Omron CX-Programmer project 新工程 (CX-Programmer 9.73)

# PLC 新PLC1: CPM2* 

## Global symbols (name address type ; comment)
0.11 BOOL  ; �0网�╈�?w�!
10.02 BOOL  ; �6�镧诜z鼯�u靑
11.01 BOOL  ; $?St$Bk?_#[2] / 粋龠诛�� / 顯�(鰟$?St$Bk?_#[2]
11.13 BOOL  ; �*�{得�逌A� �69
13.04 BOOL  ; 制动
13.05 BOOL  ; �东嚼浯�
13.13 BOOL  ; /站齴遅喵顎^
13.14 BOOL  ; '@� nK瞈�饾y�4
15.07 BOOL  ; 獱^践蒘��揧PB�
1.11 BOOL  ; �膈g�e稞��濨5
25.13 BOOL  ; 
2.07 BOOL  ; 4╖�铴�煙呀腩
31.11 BOOL  ; �愴�搡k賴�$欈]
43.02 BOOL  ; 抆葵`|%���A
4.02 BOOL  ; 啐-�旜��FA
6.01 BOOL  ; 卟_�垤��巻(埨O
6.09 BOOL  ; 蓮7挑��┹茒Q
6.13 BOOL  ; 珴;埗�符�禞�b
AR4.01 BOOL  ; _�/頡骫鹐y�a
LR12.14 BOOL  ; �$_Y般鬻锟絸�>
LR13.11 BOOL  ; 慊纂��}煂l 棝v
LR9.05 BOOL  ; J荦�~Mw�	k

## Program 新程序1 (no task)
; 这个PLC程序实现了一个锰钢生产线的控制系统，应用于钢铁厂的锰钢生产工艺。 / 系统包含启动按钮、停止按钮、手动/自动开关、加热炉温度传感器、轧机压力传感器、冷却水流量传感器。 / 外部执行设备包括加热炉控制、轧机控制、冷却水泵控制、报警灯。 / 系统通过启动按钮触发整个流程，随后激活加热炉控制对锰钢原料进行加热。在加热完成后，系统启动轧机控制对原料进行轧制成型。特别地，加热炉控制和轧机控制不可同时启动，以避免设备间的冲突，确保生产过程平稳进行。按下加热按钮时，激活加热炉控制进行加热。按下轧制按钮时，激活轧机控制进行轧制。轧制完成后，启动冷却水泵控制对钢材进行冷却，并确保相关状态正常。启动按钮按下时，激活冷却水泵控制进行冷却。冷却水流量传感器正常时，维持冷却水泵控制的运行。 / 操作员可以通过手动/自动切换开关选择运行模式。在手动模式下，按下手动模式按钮置位手动模式标志，随后通过按钮控制加热炉控制、轧机控制和冷却水泵控制。在自动模式下，按下自动模式按钮置位自动模式标志，随后通过按钮触发流程。手动模式标志和自动模式标志不可同时置位，以保证模式切换的清晰性和安全性。 / 此外，如果加热炉温度传感器检测到温度超限，报警灯会立即点亮，提示操作员采取措施。加热炉温度传感器检测加热状态时，系统进入准备阶段。异常发生时，报警灯点亮提示操作员。同理，当轧机压力传感器检测到压力超出安全范围时，报警灯也会亮起，确保设备不受损。轧机压力传感器检测轧制状态时，系统继续运行。异常发生时，报警灯点亮提示操作员。系统中使用加热炉启动延时定时器 (TIM001)、轧机启动延时定时器 (TIM002) 和冷却水泵启动延时定时器 (TIM003) 控制流程的时间间隔，避免操作过快导致的故障。任何时候按下停止按钮，系统会停止部分输出，确保紧急情况下的安全。

### Section 段1

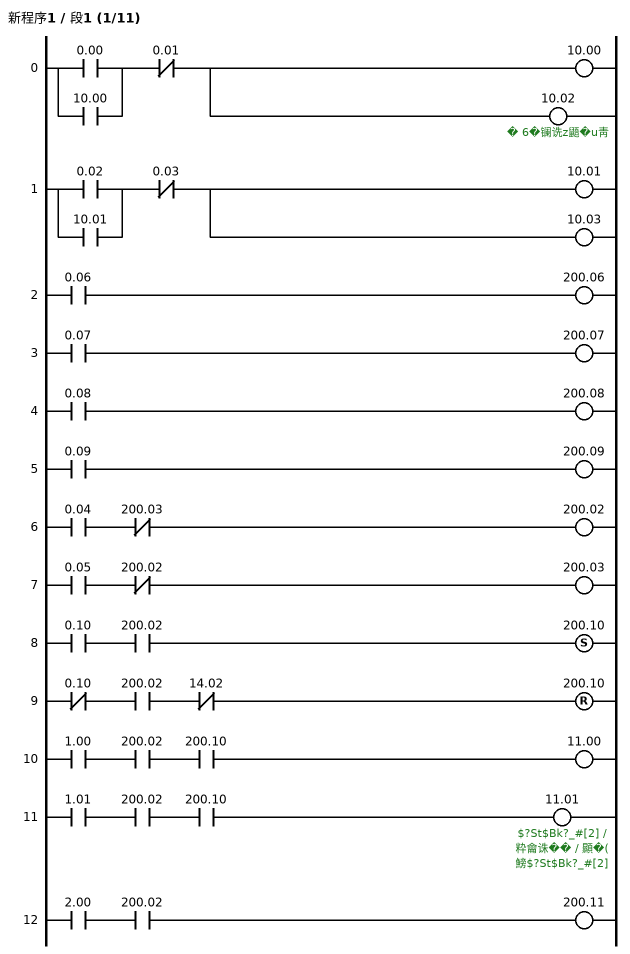
; rung 0
LD 0.00
OR 10.00
ANDNOT 0.01
OUT 10.00
OUT 10.02  ; �6�镧诜z鼯�u靑
; rung 1
LD 0.02
OR 10.01
ANDNOT 0.03
OUT 10.01
OUT 10.03
; rung 2
LD 0.06
OUT 200.06
; rung 3
LD 0.07
OUT 200.07
; rung 4
LD 0.08
OUT 200.08
; rung 5
LD 0.09
OUT 200.09
; rung 6
LD 0.04
ANDNOT 200.03
OUT 200.02
; rung 7
LD 0.05
ANDNOT 200.02
OUT 200.03
; rung 8
LD 0.10
AND 200.02
SET 200.10
; rung 9
LDNOT 0.10
AND 200.02
ANDNOT 14.02
RSET 200.10
; rung 10
LD 1.00
AND 200.02
AND 200.10
OUT 11.00
; rung 11
LD 1.01
AND 200.02
AND 200.10
OUT 11.01  ; $?St$Bk?_#[2] / 粋龠诛�� / 顯�(鰟$?St$Bk?_#[2]
; rung 12
LD 2.00
AND 200.02
OUT 200.11

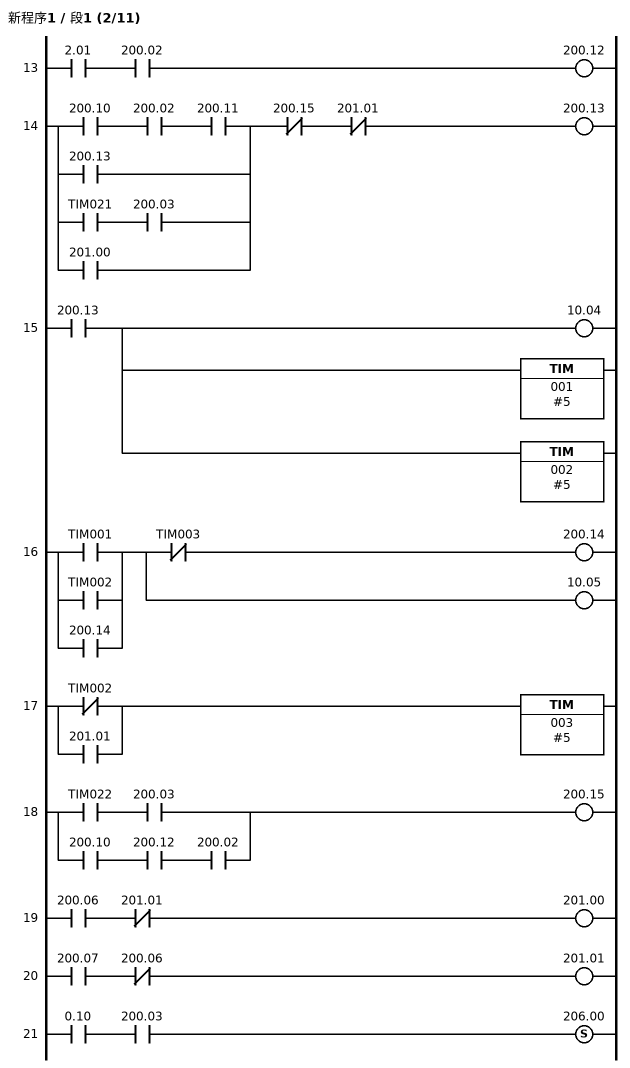
; rung 13
LD 2.01
AND 200.02
OUT 200.12
; rung 14
LD 200.10
AND 200.02
AND 200.11
OR 200.13
LD TIM021
AND 200.03
ORLD
OR 201.00
ANDNOT 200.15
ANDNOT 201.01
OUT 200.13
; rung 15
LD 200.13
OUT 10.04
TIM 001 #5
TIM 002 #5
; rung 16
LD TIM001
OR TIM002
OR 200.14
OUT TR0
ANDNOT TIM003
OUT 200.14
LD TR0
OUT 10.05
; rung 17
LDNOT TIM002
OR 201.01
TIM 003 #5
; rung 18
LD TIM022
AND 200.03
LD 200.10
AND 200.12
AND 200.02
ORLD
OUT 200.15
; rung 19
LD 200.06
ANDNOT 201.01
OUT 201.00
; rung 20
LD 200.07
ANDNOT 200.06
OUT 201.01
; rung 21
LD 0.10
AND 200.03
SET 206.00

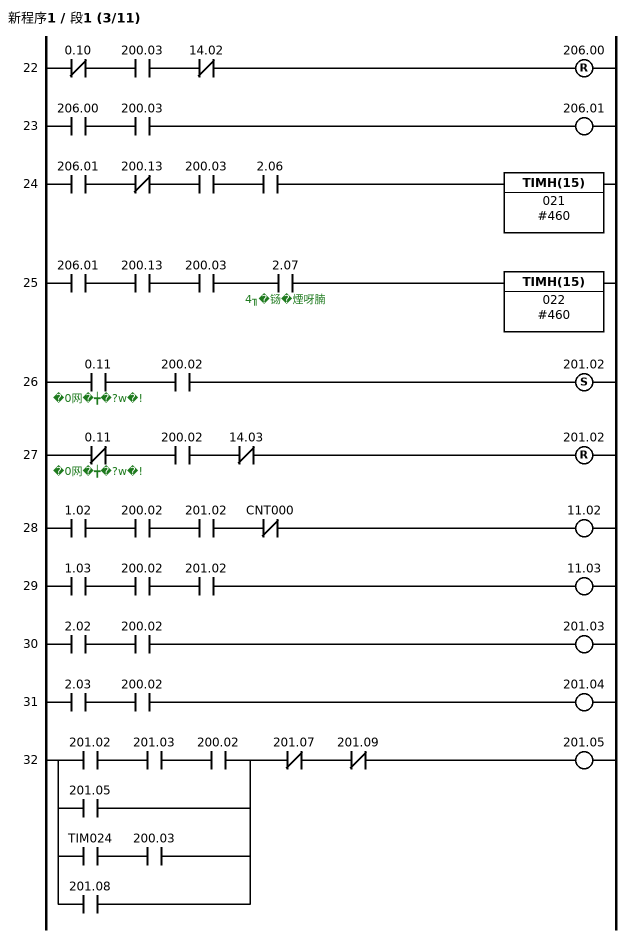
; rung 22
LDNOT 0.10
AND 200.03
ANDNOT 14.02
RSET 206.00
; rung 23
LD 206.00
AND 200.03
OUT 206.01
; rung 24
LD 206.01
ANDNOT 200.13
AND 200.03
AND 2.06
TIMH(15) 021 #460
; rung 25
LD 206.01
AND 200.13
AND 200.03
AND 2.07  ; 4╖�铴�煙呀腩
TIMH(15) 022 #460
; rung 26
LD 0.11  ; �0网�╈�?w�!
AND 200.02
SET 201.02
; rung 27
LDNOT 0.11  ; �0网�╈�?w�!
AND 200.02
ANDNOT 14.03
RSET 201.02
; rung 28
LD 1.02
AND 200.02
AND 201.02
ANDNOT CNT000
OUT 11.02
; rung 29
LD 1.03
AND 200.02
AND 201.02
OUT 11.03
; rung 30
LD 2.02
AND 200.02
OUT 201.03
; rung 31
LD 2.03
AND 200.02
OUT 201.04
; rung 32
LD 201.02
AND 201.03
AND 200.02
OR 201.05
LD TIM024
AND 200.03
ORLD
OR 201.08
ANDNOT 201.07
ANDNOT 201.09
OUT 201.05

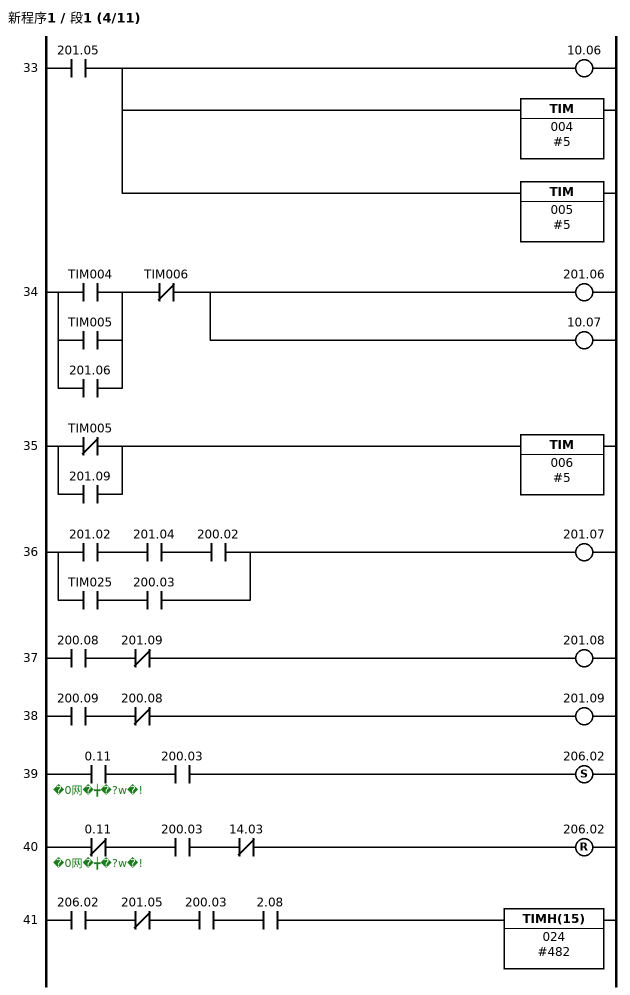
; rung 33
LD 201.05
OUT 10.06
TIM 004 #5
TIM 005 #5
; rung 34
LD TIM004
OR TIM005
OR 201.06
ANDNOT TIM006
OUT 201.06
OUT 10.07
; rung 35
LDNOT TIM005
OR 201.09
TIM 006 #5
; rung 36
LD 201.02
AND 201.04
AND 200.02
LD TIM025
AND 200.03
ORLD
OUT 201.07
; rung 37
LD 200.08
ANDNOT 201.09
OUT 201.08
; rung 38
LD 200.09
ANDNOT 200.08
OUT 201.09
; rung 39
LD 0.11  ; �0网�╈�?w�!
AND 200.03
SET 206.02
; rung 40
LDNOT 0.11  ; �0网�╈�?w�!
AND 200.03
ANDNOT 14.03
RSET 206.02
; rung 41
LD 206.02
ANDNOT 201.05
AND 200.03
AND 2.08
TIMH(15) 024 #482

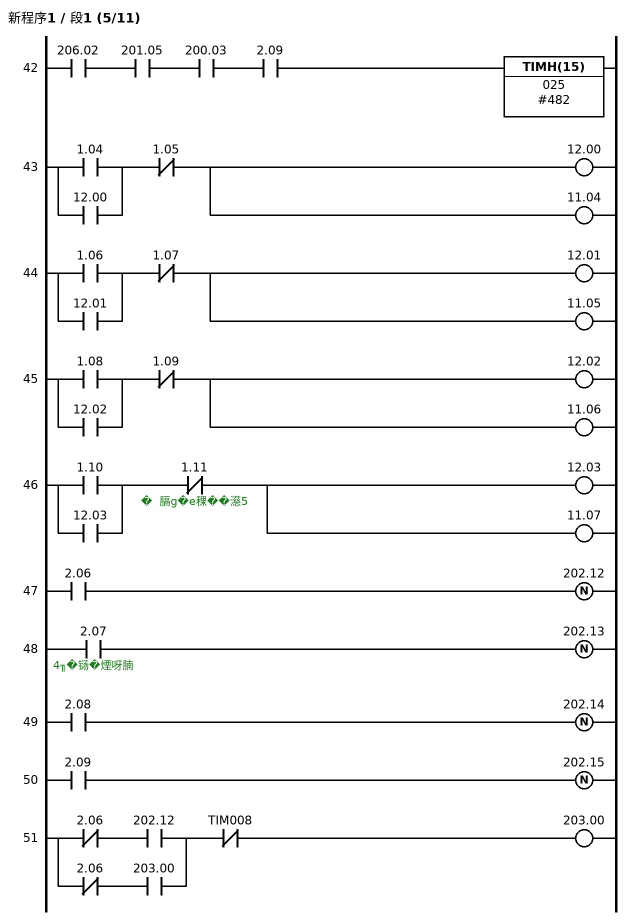
; rung 42
LD 206.02
AND 201.05
AND 200.03
AND 2.09
TIMH(15) 025 #482
; rung 43
LD 1.04
OR 12.00
ANDNOT 1.05
OUT 12.00
OUT 11.04
; rung 44
LD 1.06
OR 12.01
ANDNOT 1.07
OUT 12.01
OUT 11.05
; rung 45
LD 1.08
OR 12.02
ANDNOT 1.09
OUT 12.02
OUT 11.06
; rung 46
LD 1.10
OR 12.03
ANDNOT 1.11  ; �膈g�e稞��濨5
OUT 12.03
OUT 11.07
; rung 47
LD 2.06
DIFD(14) 202.12
; rung 48
LD 2.07  ; 4╖�铴�煙呀腩
DIFD(14) 202.13
; rung 49
LD 2.08
DIFD(14) 202.14
; rung 50
LD 2.09
DIFD(14) 202.15
; rung 51
LDNOT 2.06
AND 202.12
LDNOT 2.06
AND 203.00
ORLD
ANDNOT TIM008
OUT 203.00

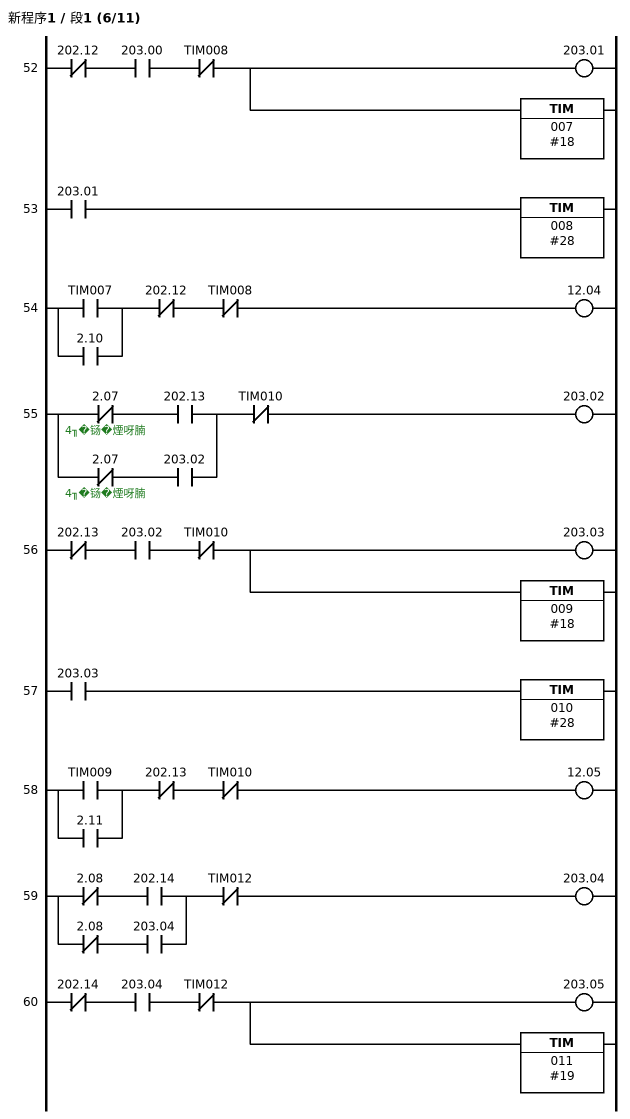
; rung 52
LDNOT 202.12
AND 203.00
ANDNOT TIM008
OUT 203.01
TIM 007 #18
; rung 53
LD 203.01
TIM 008 #28
; rung 54
LD TIM007
OR 2.10
ANDNOT 202.12
ANDNOT TIM008
OUT 12.04
; rung 55
LDNOT 2.07  ; 4╖�铴�煙呀腩
AND 202.13
LDNOT 2.07  ; 4╖�铴�煙呀腩
AND 203.02
ORLD
ANDNOT TIM010
OUT 203.02
; rung 56
LDNOT 202.13
AND 203.02
ANDNOT TIM010
OUT 203.03
TIM 009 #18
; rung 57
LD 203.03
TIM 010 #28
; rung 58
LD TIM009
OR 2.11
ANDNOT 202.13
ANDNOT TIM010
OUT 12.05
; rung 59
LDNOT 2.08
AND 202.14
LDNOT 2.08
AND 203.04
ORLD
ANDNOT TIM012
OUT 203.04
; rung 60
LDNOT 202.14
AND 203.04
ANDNOT TIM012
OUT 203.05
TIM 011 #19

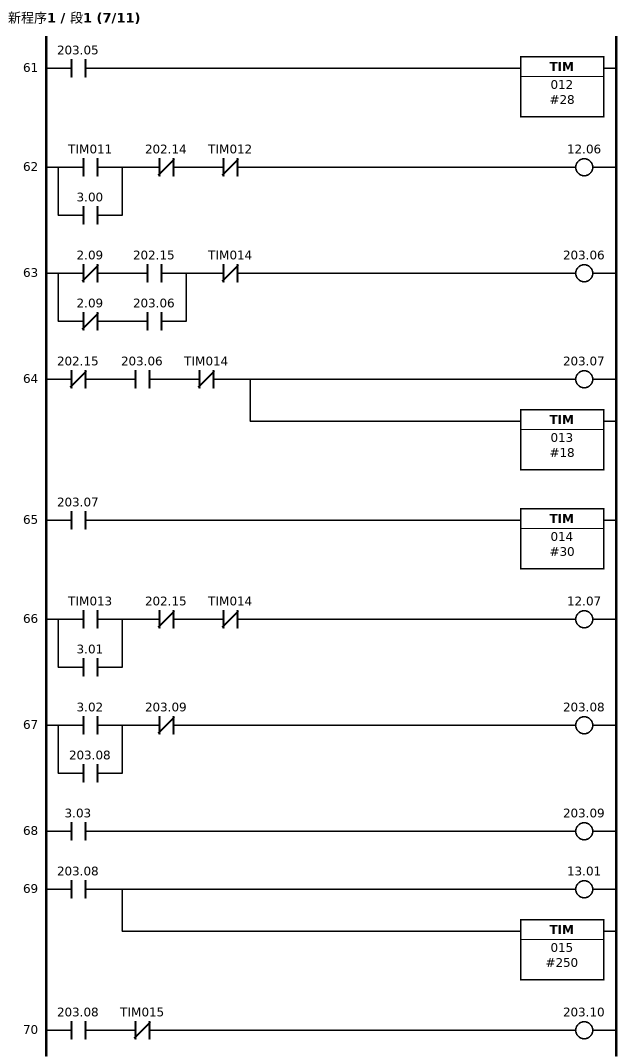
; rung 61
LD 203.05
TIM 012 #28
; rung 62
LD TIM011
OR 3.00
ANDNOT 202.14
ANDNOT TIM012
OUT 12.06
; rung 63
LDNOT 2.09
AND 202.15
LDNOT 2.09
AND 203.06
ORLD
ANDNOT TIM014
OUT 203.06
; rung 64
LDNOT 202.15
AND 203.06
ANDNOT TIM014
OUT 203.07
TIM 013 #18
; rung 65
LD 203.07
TIM 014 #30
; rung 66
LD TIM013
OR 3.01
ANDNOT 202.15
ANDNOT TIM014
OUT 12.07
; rung 67
LD 3.02
OR 203.08
ANDNOT 203.09
OUT 203.08
; rung 68
LD 3.03
OUT 203.09
; rung 69
LD 203.08
OUT 13.01
TIM 015 #250
; rung 70
LD 203.08
ANDNOT TIM015
OUT 203.10

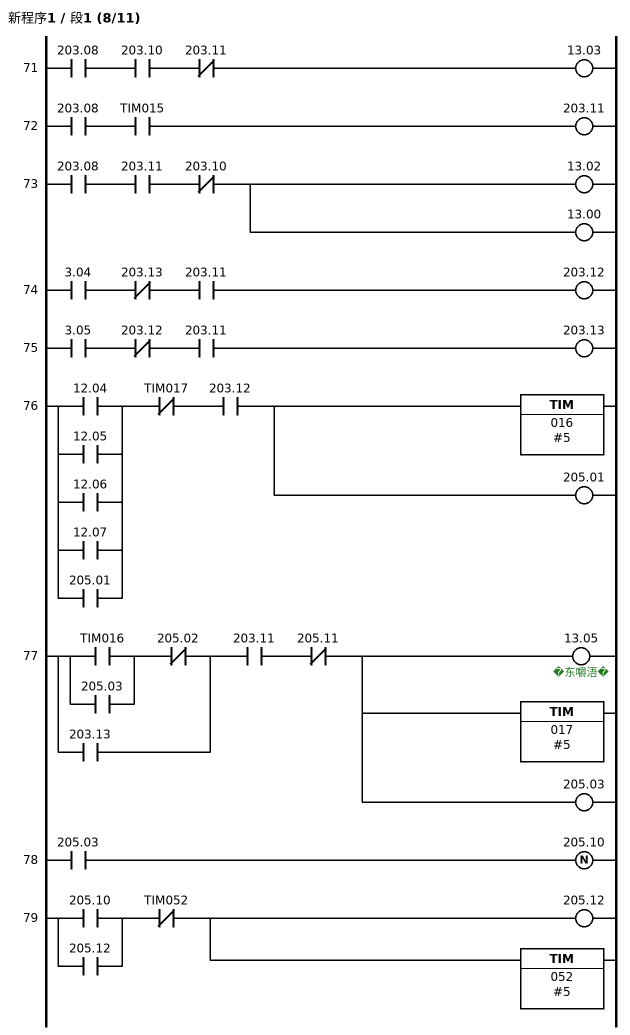
; rung 71
LD 203.08
AND 203.10
ANDNOT 203.11
OUT 13.03
; rung 72
LD 203.08
AND TIM015
OUT 203.11
; rung 73
LD 203.08
AND 203.11
ANDNOT 203.10
OUT 13.02
OUT 13.00
; rung 74
LD 3.04
ANDNOT 203.13
AND 203.11
OUT 203.12
; rung 75
LD 3.05
ANDNOT 203.12
AND 203.11
OUT 203.13
; rung 76
LD 12.04
OR 12.05
OR 12.06
OR 12.07
OR 205.01
ANDNOT TIM017
AND 203.12
TIM 016 #5
OUT 205.01
; rung 77
LD TIM016
OR 205.03
ANDNOT 205.02
OR 203.13
AND 203.11
ANDNOT 205.11
OUT 13.05  ; �东嚼浯�
TIM 017 #5
OUT 205.03
; rung 78
LD 205.03
DIFD(14) 205.10
; rung 79
LD 205.10
OR 205.12
ANDNOT TIM052
OUT 205.12
TIM 052 #5

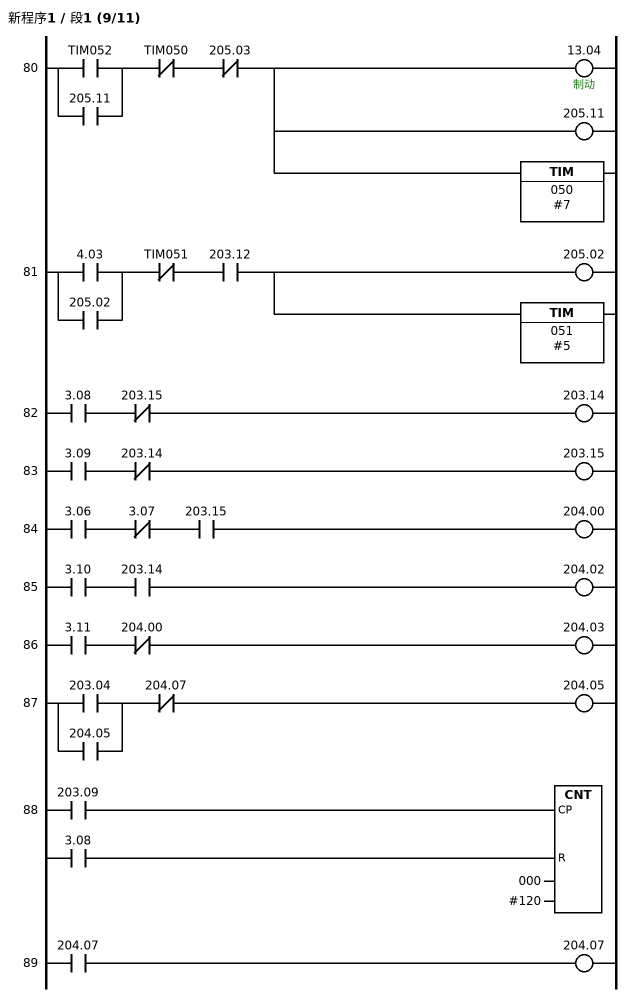
; rung 80
LD TIM052
OR 205.11
ANDNOT TIM050
ANDNOT 205.03
OUT 13.04  ; 制动
OUT 205.11
TIM 050 #7
; rung 81
LD 4.03
OR 205.02
ANDNOT TIM051
AND 203.12
OUT 205.02
TIM 051 #5
; rung 82
LD 3.08
ANDNOT 203.15
OUT 203.14
; rung 83
LD 3.09
ANDNOT 203.14
OUT 203.15
; rung 84
LD 3.06
ANDNOT 3.07
AND 203.15
OUT 204.00
; rung 85
LD 3.10
AND 203.14
OUT 204.02
; rung 86
LD 3.11
ANDNOT 204.00
OUT 204.03
; rung 87
LD 203.04
OR 204.05
ANDNOT 204.07
OUT 204.05
; rung 88
LD 203.09
LD 3.08
CNT 000 #120
; rung 89
LD 204.07
OUT 204.07

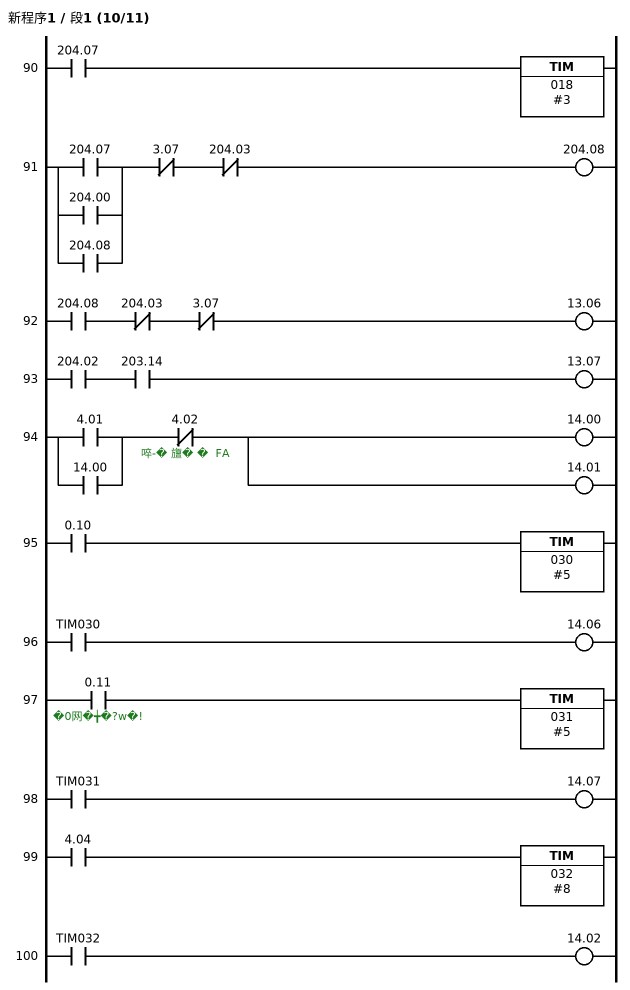
; rung 90
LD 204.07
TIM 018 #3
; rung 91
LD 204.07
OR 204.00
OR 204.08
ANDNOT 3.07
ANDNOT 204.03
OUT 204.08
; rung 92
LD 204.08
ANDNOT 204.03
ANDNOT 3.07
OUT 13.06
; rung 93
LD 204.02
AND 203.14
OUT 13.07
; rung 94
LD 4.01
OR 14.00
ANDNOT 4.02  ; 啐-�旜��FA
OUT 14.00
OUT 14.01
; rung 95
LD 0.10
TIM 030 #5
; rung 96
LD TIM030
OUT 14.06
; rung 97
LD 0.11  ; �0网�╈�?w�!
TIM 031 #5
; rung 98
LD TIM031
OUT 14.07
; rung 99
LD 4.04
TIM 032 #8
; rung 100
LD TIM032
OUT 14.02

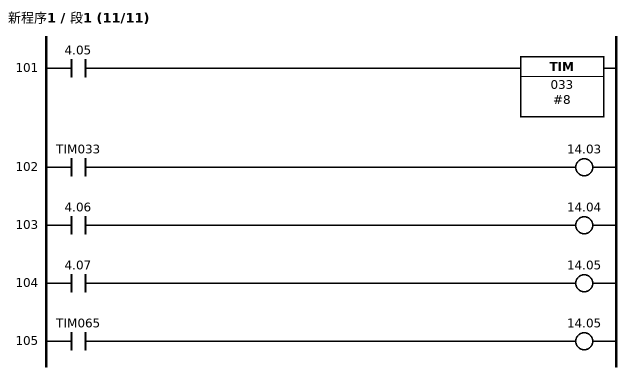
; rung 101
LD 4.05
TIM 033 #8
; rung 102
LD TIM033
OUT 14.03
; rung 103
LD 4.06
OUT 14.04
; rung 104
LD 4.07
OUT 14.05
; rung 105
LD TIM065
OUT 14.05
; rung 106
END(01)